Omron Sysmac Studio project Tp last version 30.20h (Comentado) (Sysmac Studio 1.54.0.64019, StandardProject)

# Controller new_Controller_0: NX1P2-9B24DT1 version 1.42
Task PrimaryTask (priority 4, period or condition 4000): Program0
Library OEN_Communication_V1_0_22 1.0.22 (contents left out)

VAR_GLOBAL
    trama : ARRAY[0..4] OF OEN\Modbus\sModbusReq := [(Enable := True, NodeAdr := 1, FunctionCode := Fn15_WriteMultipleCoils, Read := (StartAddressRemote := 0, StartAddressLocal := 0, Count := 0), Write := (StartAddressRemote := 0, StartAddressLocal := 0, Count := 80)), (Enable := True, NodeAdr := 1, FunctionCode := Fn02_ReadDiscreteInputs, Read := (StartAddressRemote := 0, StartAddressLocal := 0, Count := 80), Write := (StartAddressRemote := 0, StartAddressLocal := 0, Count := 0)), (Enable := True, NodeAdr := 1, FunctionCode := Fn04_ReadInputRegisters, Read := (StartAddressRemote := 0, StartAddressLocal := 0, Count := 25), Write := (StartAddressRemote := 0, StartAddressLocal := 0, Count := 0)), (Enable := True, NodeAdr := 1, FunctionCode := Fn16_WriteMultipleRegisters, Read := (StartAddressRemote := 0, StartAddressLocal := 0, Count := 0), Write := (StartAddressRemote := 0, StartAddressLocal := 0, Count := 25)), (Enable := False, NodeAdr := 0, FunctionCode := Fn01_ReadCoils, Read := (StartAddressRemote := 0, StartAddressLocal := 0, Count := 0), Write := (StartAddressRemote := 0, StartAddressLocal := 0, Count := 0))];  (* Trama Responsável pelo invio de informação; published *)
END_VAR
VAR_GLOBAL RETAIN
    Dig_Outputs AT %D10 : ARRAY[0..100] OF BOOL;  (* Digital Outputs; published *)
    Dig_Inputs AT %D20 : ARRAY[0..100] OF BOOL;  (* Digital Inputs; published *)
    Anal_Outputs AT %D30 : ARRAY[0..25] OF WORD;  (* Analog Outputs; published *)
    Anal_Inputs AT %D55 : ARRAY[0..25] OF WORD;  (* Analog Inputs; published *)
END_VAR
VAR_GLOBAL
    Start : BOOL;  (* Acionamento sistema; at BuiltInIO://cpu/#0/Input_Bit_00 *)
    Stop : BOOL;  (* Paragem Sistema; at BuiltInIO://cpu/#0/Input_Bit_01 *)
    ledstart : BOOL;  (* Sinal luminoso de acionamento sistema; at BuiltInIO://cpu/#0/Output_Bit_00 *)
    Colocar : BOOL;  (* Botão Colocar Stacker; at BuiltInIO://cpu/#0/Input_Bit_02 *)
    Remover : BOOL;  (* Botão Remover Stacker; at BuiltInIO://cpu/#0/Input_Bit_03 *)
    NovaCaixa : BOOL;  (* Botão Nova Caixa; at BuiltInIO://cpu/#0/Input_Bit_04 *)
    ledstop : BOOL;  (* Sinal luminoso de paragem sistema; at BuiltInIO://cpu/#0/Output_Bit_01 *)
    ledcolocar : BOOL;  (* Sinal luminoso colocação caixa; at BuiltInIO://cpu/#0/Output_Bit_02 *)
    ledremover : BOOL;  (* Sinal luminoso remoção caixa; at BuiltInIO://cpu/#0/Output_Bit_03 *)
END_VAR

PROGRAM Program0
VAR RETAIN
    Etapas AT %D0 : INT := 0;  (* This variable is change current phase *)
END_VAR
VAR
    Communication_Factory : OEN\Modbus\ModbusTCP_Client;
    Timer2s : TON;
END_VAR
VAR RETAIN
    VariableAux AT %D1 : WORD;  (* Var.aux Medidor Altura 1 *)
END_VAR
VAR
    Timer1 : TON;
    Time_Aux_5 : TIME;  (* Timer_Aux_5s *)
    Timer4 : TON;
    Timer5 : TON;
    Timevariavel : TIME;
    Timer6 : TON;
    Timer10s : TON;
    Timer7 : TON;
    Timer8 : TON;
    Timer9 : TON;
END_VAR
VAR RETAIN
    VariableAux2 : WORD;  (* Var.aux Medidor Altura 1 *)
END_VAR
VAR
    Time_Aux_20 : TIME;  (* Timer_Aux_20s *)
    Timer20 : TON;
    Timer21 : TON;
    Time_Aux_21 : TIME;
    Timer30 : TON;
    Timer31 : TON;
    Timer32 : TON;
    Timer33 : TON;
    Timer34 : TON;
    Timer35 : TON;
    Timer36 : TON;
    Timer37 : TON;
    Timer38 : TON;
    Timer2 : TON;
    Timer2p : TON;
    Timer101 : TON;
    Timer3p : TON;
END_VAR
VAR RETAIN
    VariavelAux10 : WORD;  (* Aux10 *)
END_VAR
VAR
    Timer4sec : TON;
    Timer4P6sec : TON;
    Timer4PPsec : TON;
    Timer5PPsec : TON;
    Timer6PPsec : TON;
    Timer7PPsec : TON;
    Timer8PPsec : TON;
    Timer9PPsec : TON;
    Timer101PPsec : TON;
    Timer10PPsec : TON;
    Timercount : TON;
    Timer3s : TON;
END_VAR
VAR RETAIN
    Count_Caixa_L : INT := 0;  (* Contador Caixa L *)
END_VAR
VAR
    Analogico_L : WORD;  (* Valor Analogico L *)
END_VAR
VAR RETAIN
    Count_Caixa_S : INT := 0;  (* Contador Caixa S *)
END_VAR
VAR
    Analogico_S : WORD;  (* Valor Analogico S *)
END_VAR
VAR RETAIN
    Count_Caixa_M : INT := 0;  (* Contador Caixa M *)
END_VAR
VAR
    Analogico_M : WORD;  (* Valor Analogico M *)
END_VAR
VAR RETAIN
    Contador_Stacker_2 : INT := 0;  (* Contador Posição Stacker 2 *)
    Analogico_Postacker2 : WORD;  (* Variavel Analogica Posição *)
END_VAR
VAR
    Timer30s : TON;
    Timer31s : TON;
    Timer32s : TON;
    TimerEsp : TON;
    TimerDecisão : TON;
    TimerDecisão2 : TON;
    Timerteste : TON;
    led : BOOL;
END_VAR
VAR_EXTERNAL
    trama : ARRAY[0..4] OF OEN\Modbus\sModbusReq;  (* Trama que envia informação *)
    dig_outputs : ARRAY[0..100] OF BOOL;  (* Digital outputs; [8] Tapete 1; [1] Led Botão 1; [2] LED Botão Start; [5] Emissor Caixa; [6] Emissor Paletes 1; [7] Emissor Paletes 2; [11] Tapete 4; [24] Esteira Transportada 11; [14] Tapete Peso (+); [17] Esteira Transportadora 2; [25] Esteira Transportadora 12; [18] Esteira Transportadora 3; [26] Esteira Transportadora 13; [16] Esteira Transportadora 1; [10] Tapete 3; [33] Two-Axis Pick &amp; Place 1 Z; [36] Two-Axis Pick &amp; Place 1 (Grab); [38] Two-Axis Pick &amp; Place 1 Rotate CW; [9] Tapete 2; [32] Two-Axis Pick &amp; Place 1 X; [41] Two-Axis Pick &amp; Place 1 Rotate CCW; [19] Esteira Transportadora 4; [20] Esteira Transportadora 5; [21] Esteira Transportadora 6; [22] Esteira Transportadora 7; [23] Esteira Transportadora 8; [30] pusher 1; [12] Tapete 5; [15] Tapete peso 2; [13] Tapete 6; [49] Stacker Crane 3(left); [47] Stacker Crane 3 lift; [54] Led Colocar; [51] Stacker Crane 3 Right ; [55] LED Remover; [53] Remover 3; [35] Two-Axis Pick &amp; Place 2 Z; [37] Two-Axis Pick &amp; Place 2 (Grab); [39] Two-Axis Pick &amp; Place 2 Rotate CW; [34] Two-Axis Pick &amp; Place 2 X; [43] Two-Axis Pick &amp; Place 1 Rotate CCW; [27] Esteira Transportadora 14; [28] Esteira Transportadora 15; [29] Esteira Transportadora 16; [31] Pusher 2; [48] Stacker Crane 1 left; [46] Stacker Crane 1 lift; [50] stacker crane 1 right; [3] LED Botão Stop *)
    dig_inputs : ARRAY[0..100] OF BOOL;  (* Digital inputs; [2] Sensor Detetar caixas; [0] Botão Start; [13] Sensor Difuso 10; [22] Sensor Difuso 19; [3] Sensor Difuso 1; [14] Sensor Difuso 11; [9] Sensor Difuso 6; [21] Sensor difuso 18; [15] Sensor Difuso 12; [16] Sensor difuso 13; [59] Sensor Difuso 27; [23] Sensor Difuso 20; [24] Sensor Difuso 21; [4] Sensor Difuso 2; [5] Sensor Difuso 3; [52] Two-Axis Pick &amp; Place 1 (Moving Z); [36] Two-Axis Pick &amp; Place 1 (Grab); [50] Two-Axis Pick &amp; Place 1 (Detected); [17] Sensor difuso 14; [18] Sensor difuso 15; [19] sensor difuso 16; [20] Sensor Difuso 17; [35] Pusher frontal; [7] Sensor Difuso 4; [8] Sensor Difuso 8; [60] Sensor Difuso 28; [29] Sensor Refletivo 1; [61] Botão Colocar; [44] Stacker Crane 3 left limit; [48] Stacker Crane 3 Middle Limit; [46] Stacker Crane 3 Right Limit; [62] Botão Remover; [31] Sensor Refletivo 3; [30] Sensor Difuso 29; [10] Sensor difuso 7; [12] Sensor Difuso 9; [26] Sensor Difuso 23; [27] Sensor Difuso 24; [32] Sensor Refletivo 4; [28] Sensor Difuso 25; [11] Sensor Difuso 8; [54] detected; [43] Stacker Crane 1 left Limit; [47] stacker Crane 1 Middle Limit; [45] Stacker Crane 1 Right Limit; [1] Botão Stop; [63] Botão Nova Caixa *)
    anal_inputs : ARRAY[0..25] OF WORD;  (* Analog inputs; [2] Balança 1 Peso (V); [1] Medidor Altura 2; [0] Medidor Altura 1; [3] Peso 2 *)
    anal_outputs : ARRAY[0..25] OF WORD;  (* Analog outputs; [2] Esteira Transportadora 9; [10] Display 1; [12] Display 3; [1] Posição 2; [11] Display 2; [6] Loading Convoyer 1; [0] Posição1 *)
    Start : BOOL;
    Stop : BOOL;
    ledstart : BOOL;
    ledstop : BOOL;
    NovaCaixa : BOOL;
    Colocar : BOOL;
    Remover : BOOL;
    ledremover : BOOL;
    ledcolocar : BOOL;
END_VAR
VAR
    _p1 : BOOL;
    _e2 : R_TRIG;
    _p3 : BOOL;
    _p4 : BOOL;
    _p5 : BOOL;
    _e6 : R_TRIG;
    _e7 : R_TRIG;
    _e8 : R_TRIG;
END_VAR

(* Section Phases: ladder, written here as Structured Text *)

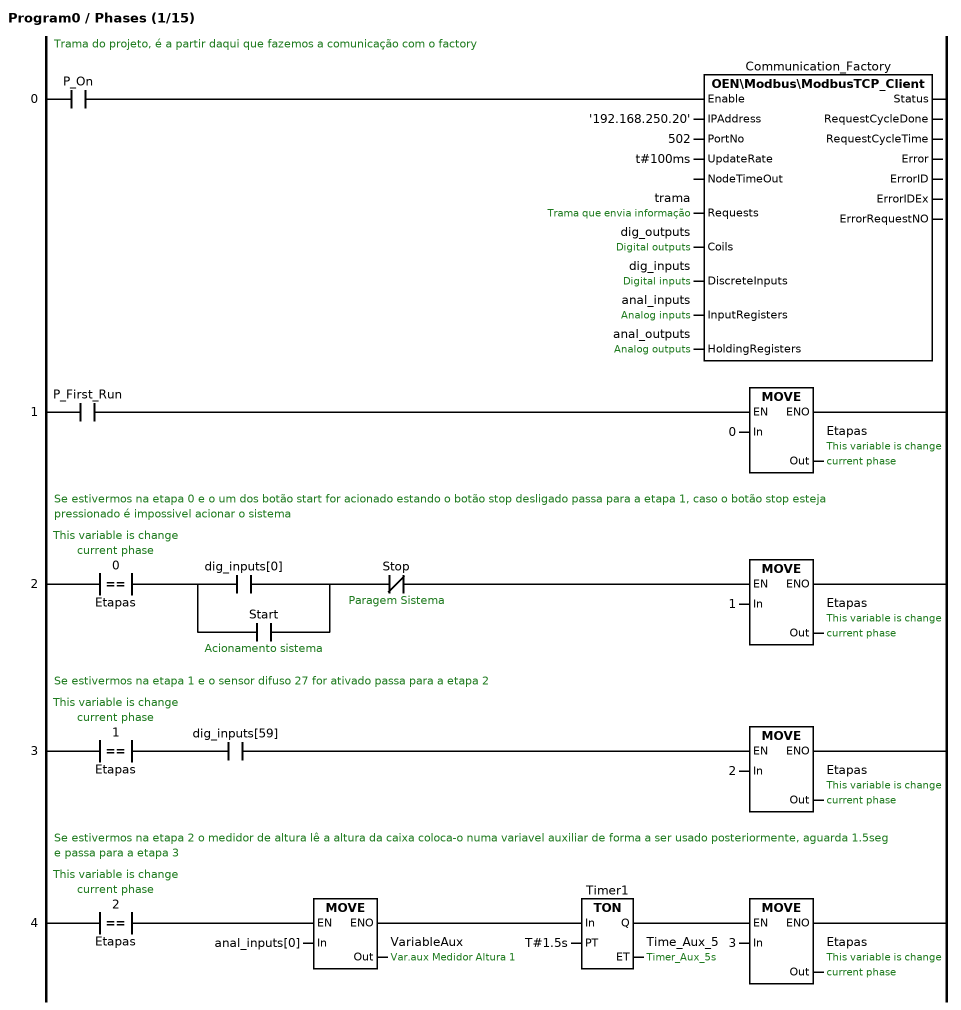
(* Rung 0: Trama do projeto, é a partir daqui que fazemos a comunicação com o factory *)
Communication_Factory(Enable := P_On, IPAddress := '192.168.250.20', PortNo := 502, UpdateRate := t#100ms, Requests := trama, Coils := dig_outputs, DiscreteInputs := dig_inputs, InputRegisters := anal_inputs, HoldingRegisters := anal_outputs);
(* Rung 1 *)
IF P_First_Run THEN Etapas := 0; END_IF;
(* Rung 2: Se estivermos na etapa 0 e o um dos botão start for acionado estando o botão stop desligado passa para a etapa 1, caso o botão stop esteja pressionado é impossivel acionar o sistema *)
IF (0 = Etapas) AND (dig_inputs[0] OR Start) AND NOT Stop THEN Etapas := 1; END_IF;
(* Rung 3: Se estivermos na etapa 1 e o sensor difuso 27 for ativado passa para a etapa 2 *)
IF (1 = Etapas) AND dig_inputs[59] THEN Etapas := 2; END_IF;
(* Rung 4: Se estivermos na etapa 2 o medidor de altura lê a altura da caixa coloca-o numa variavel auxiliar de forma a ser usado posteriormente, aguarda 1.5seg e passa para a etapa 3 *)
IF 2 = Etapas THEN VariableAux := anal_inputs[0]; END_IF;
Timer1(In := 2 = Etapas, PT := T#1.5s, ET => Time_Aux_5);
IF Timer1.Q THEN Etapas := 3; END_IF;

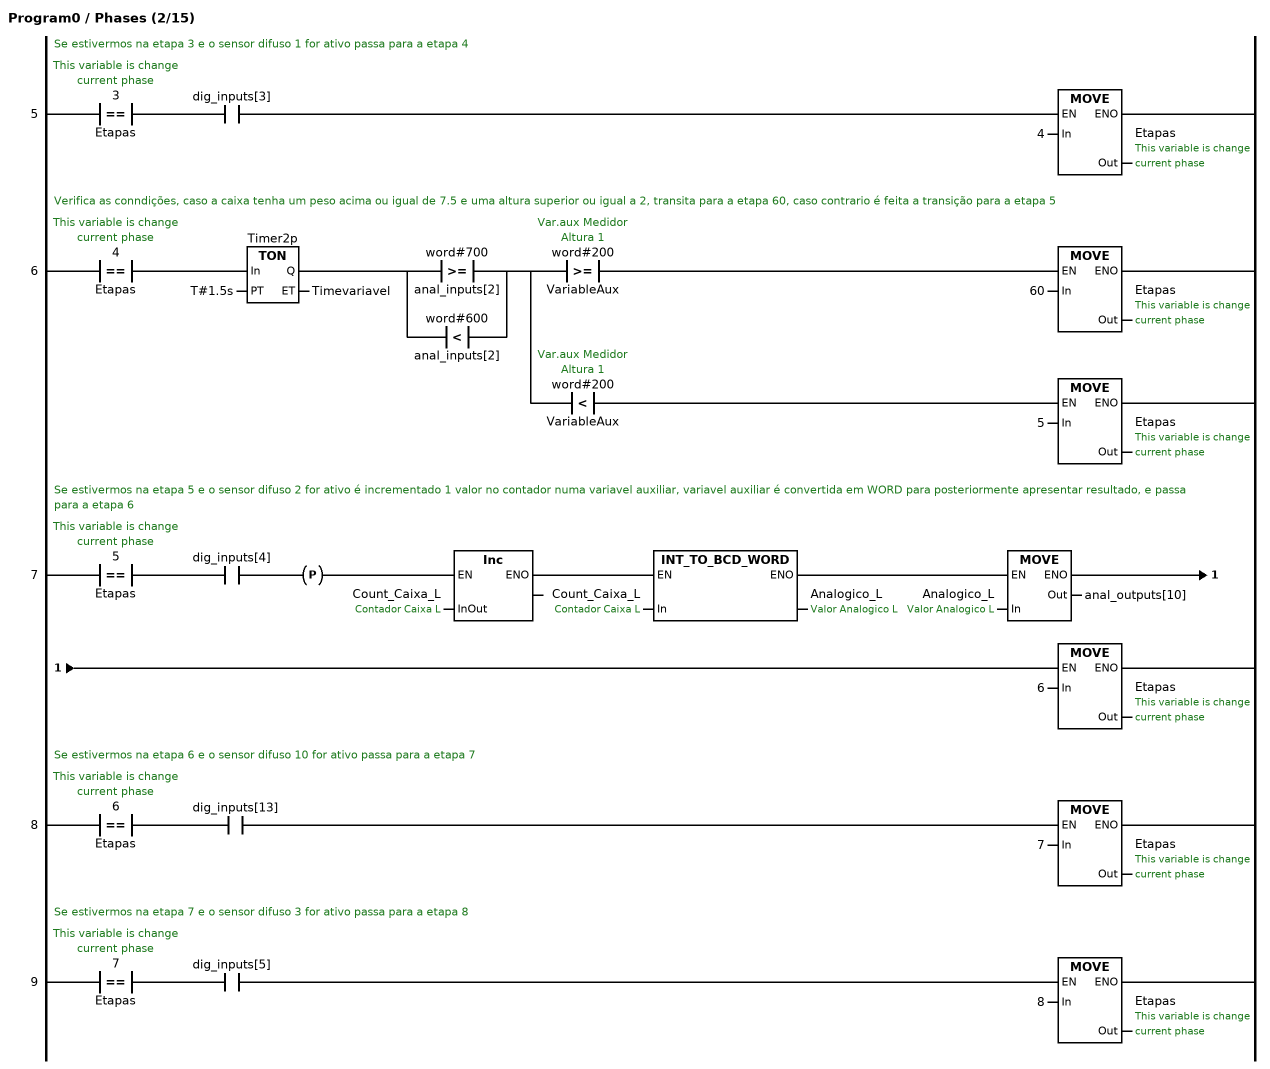
(* Rung 5: Se estivermos na etapa 3 e o sensor difuso 1 for ativo passa para a etapa 4 *)
IF (3 = Etapas) AND dig_inputs[3] THEN Etapas := 4; END_IF;
(* Rung 6: Verifica as conndições, caso a caixa tenha um peso acima ou igual de 7.5 e uma altura superior ou igual a 2, transita para a etapa 60, caso contrario é feita a transição para a etapa 5 *)
Timer2p(In := 4 = Etapas, PT := T#1.5s, ET => Timevariavel);
_p1 := Timer2p.Q AND ((word#700 >= anal_inputs[2]) OR (word#600 < anal_inputs[2]));
IF _p1 AND (word#200 >= VariableAux) THEN Etapas := 60; END_IF;
IF _p1 AND (word#200 < VariableAux) THEN Etapas := 5; END_IF;
(* Rung 7: Se estivermos na etapa 5 e o sensor difuso 2 for ativo é incrementado 1 valor no contador numa variavel auxiliar, variavel auxiliar é convertida em WORD para posteriormente apresentar resultado, e passa para a etapa 6 *)
_e2(CLK := (5 = Etapas) AND dig_inputs[4]);
IF _e2.Q THEN
    Inc(InOut := Count_Caixa_L);
    Analogico_L := INT_TO_BCD_WORD(In := Count_Caixa_L);
    anal_outputs[10] := Analogico_L;
    Etapas := 6;
END_IF;
(* Rung 8: Se estivermos na etapa 6 e o sensor difuso 10 for ativo passa para a etapa 7 *)
IF (6 = Etapas) AND dig_inputs[13] THEN Etapas := 7; END_IF;
(* Rung 9: Se estivermos na etapa 7 e o sensor difuso 3 for ativo passa para a etapa 8 *)
IF (7 = Etapas) AND dig_inputs[5] THEN Etapas := 8; END_IF;

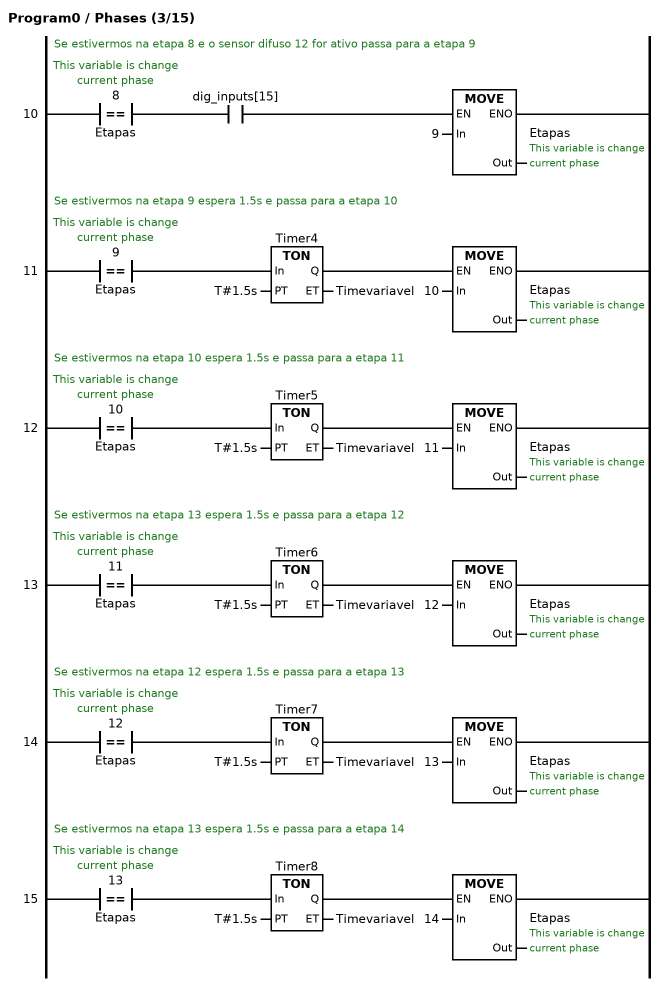
(* Rung 10: Se estivermos na etapa 8 e o sensor difuso 12 for ativo passa para a etapa 9 *)
IF (8 = Etapas) AND dig_inputs[15] THEN Etapas := 9; END_IF;
(* Rung 11: Se estivermos na etapa 9 espera 1.5s e passa para a etapa 10 *)
Timer4(In := 9 = Etapas, PT := T#1.5s, ET => Timevariavel);
IF Timer4.Q THEN Etapas := 10; END_IF;
(* Rung 12: Se estivermos na etapa 10 espera 1.5s e passa para a etapa 11 *)
Timer5(In := 10 = Etapas, PT := T#1.5s, ET => Timevariavel);
IF Timer5.Q THEN Etapas := 11; END_IF;
(* Rung 13: Se estivermos na etapa 13 espera 1.5s e passa para a etapa 12 *)
Timer6(In := 11 = Etapas, PT := T#1.5s, ET => Timevariavel);
IF Timer6.Q THEN Etapas := 12; END_IF;
(* Rung 14: Se estivermos na etapa 12 espera 1.5s e passa para a etapa 13 *)
Timer7(In := 12 = Etapas, PT := T#1.5s, ET => Timevariavel);
IF Timer7.Q THEN Etapas := 13; END_IF;
(* Rung 15: Se estivermos na etapa 13 espera 1.5s e passa para a etapa 14 *)
Timer8(In := 13 = Etapas, PT := T#1.5s, ET => Timevariavel);
IF Timer8.Q THEN Etapas := 14; END_IF;

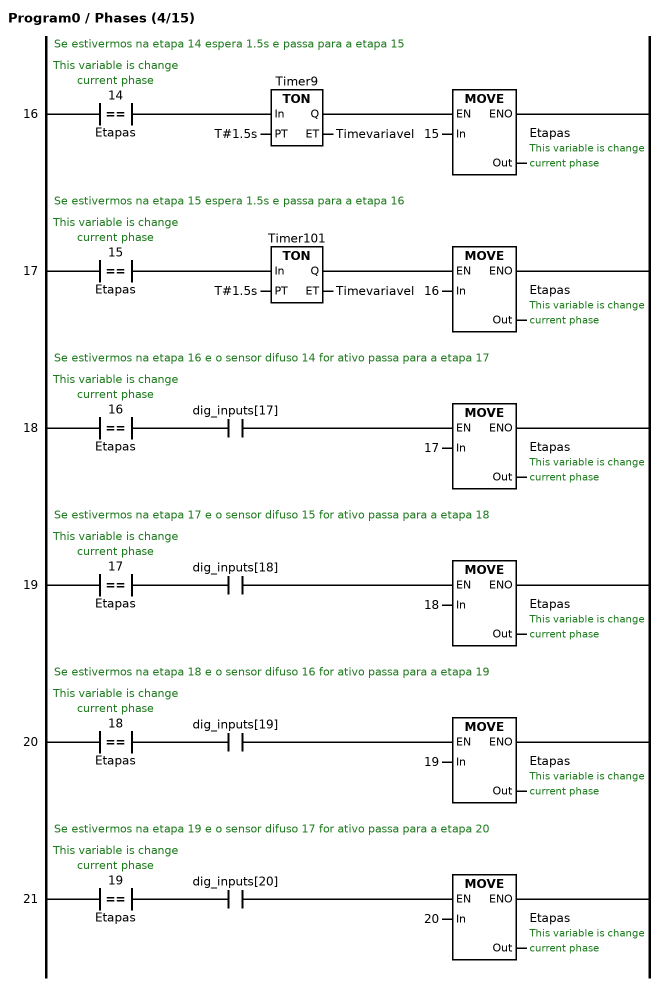
(* Rung 16: Se estivermos na etapa 14 espera 1.5s e passa para a etapa 15 *)
Timer9(In := 14 = Etapas, PT := T#1.5s, ET => Timevariavel);
IF Timer9.Q THEN Etapas := 15; END_IF;
(* Rung 17: Se estivermos na etapa 15 espera 1.5s e passa para a etapa 16 *)
Timer101(In := 15 = Etapas, PT := T#1.5s, ET => Timevariavel);
IF Timer101.Q THEN Etapas := 16; END_IF;
(* Rung 18: Se estivermos na etapa 16 e o sensor difuso 14 for ativo passa para a etapa 17 *)
IF (16 = Etapas) AND dig_inputs[17] THEN Etapas := 17; END_IF;
(* Rung 19: Se estivermos na etapa 17 e o sensor difuso 15 for ativo passa para a etapa 18 *)
IF (17 = Etapas) AND dig_inputs[18] THEN Etapas := 18; END_IF;
(* Rung 20: Se estivermos na etapa 18 e o sensor difuso 16 for ativo passa para a etapa 19 *)
IF (18 = Etapas) AND dig_inputs[19] THEN Etapas := 19; END_IF;
(* Rung 21: Se estivermos na etapa 19 e o sensor difuso 17 for ativo passa para a etapa 20 *)
IF (19 = Etapas) AND dig_inputs[20] THEN Etapas := 20; END_IF;

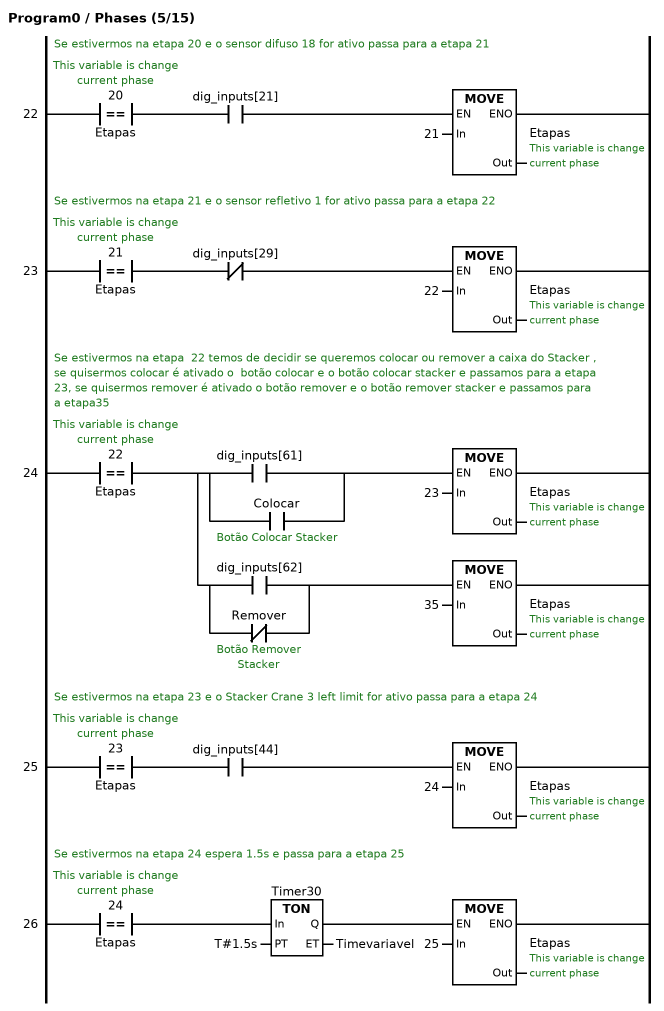
(* Rung 22: Se estivermos na etapa 20 e o sensor difuso 18 for ativo passa para a etapa 21 *)
IF (20 = Etapas) AND dig_inputs[21] THEN Etapas := 21; END_IF;
(* Rung 23: Se estivermos na etapa 21 e o sensor refletivo 1 for ativo passa para a etapa 22 *)
IF (21 = Etapas) AND NOT dig_inputs[29] THEN Etapas := 22; END_IF;
(* Rung 24: Se estivermos na etapa  22 temos de decidir se queremos colocar ou remover a caixa do Stacker , se quisermos colocar é ativado o  botão colocar e o botão colocar stacker e passamos para a etapa 23, se quisermos remover é ativado o botão remover e o botão remover stacker e passamos para a etapa35 *)
_p3 := 22 = Etapas;
IF (22 = Etapas) AND (dig_inputs[61] OR Colocar) THEN Etapas := 23; END_IF;
IF _p3 AND (dig_inputs[62] OR NOT Remover) THEN Etapas := 35; END_IF;
(* Rung 25: Se estivermos na etapa 23 e o Stacker Crane 3 left limit for ativo passa para a etapa 24 *)
IF (23 = Etapas) AND dig_inputs[44] THEN Etapas := 24; END_IF;
(* Rung 26: Se estivermos na etapa 24 espera 1.5s e passa para a etapa 25 *)
Timer30(In := 24 = Etapas, PT := T#1.5s, ET => Timevariavel);
IF Timer30.Q THEN Etapas := 25; END_IF;

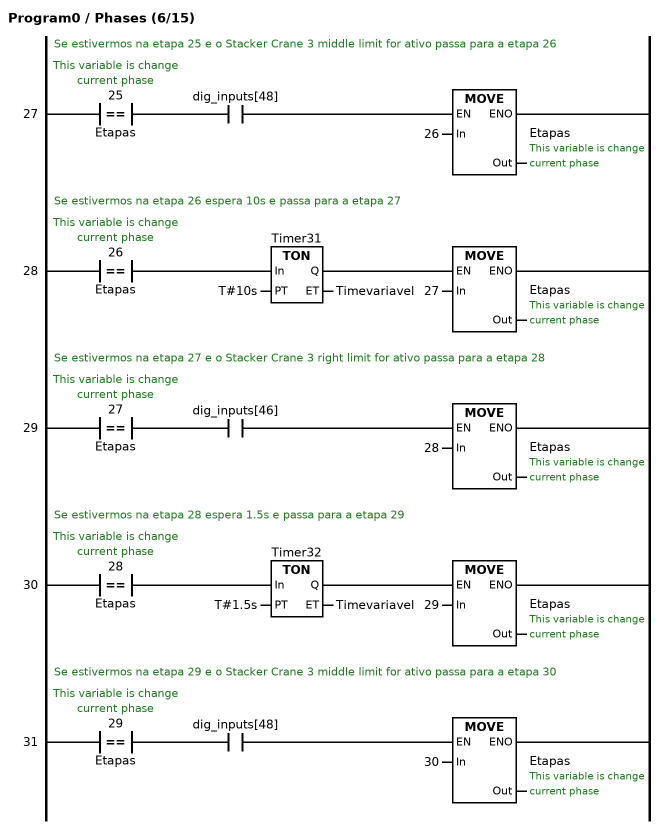
(* Rung 27: Se estivermos na etapa 25 e o Stacker Crane 3 middle limit for ativo passa para a etapa 26 *)
IF (25 = Etapas) AND dig_inputs[48] THEN Etapas := 26; END_IF;
(* Rung 28: Se estivermos na etapa 26 espera 10s e passa para a etapa 27 *)
Timer31(In := 26 = Etapas, PT := T#10s, ET => Timevariavel);
IF Timer31.Q THEN Etapas := 27; END_IF;
(* Rung 29: Se estivermos na etapa 27 e o Stacker Crane 3 right limit for ativo passa para a etapa 28 *)
IF (27 = Etapas) AND dig_inputs[46] THEN Etapas := 28; END_IF;
(* Rung 30: Se estivermos na etapa 28 espera 1.5s e passa para a etapa 29 *)
Timer32(In := 28 = Etapas, PT := T#1.5s, ET => Timevariavel);
IF Timer32.Q THEN Etapas := 29; END_IF;
(* Rung 31: Se estivermos na etapa 29 e o Stacker Crane 3 middle limit for ativo passa para a etapa 30 *)
IF (29 = Etapas) AND dig_inputs[48] THEN Etapas := 30; END_IF;

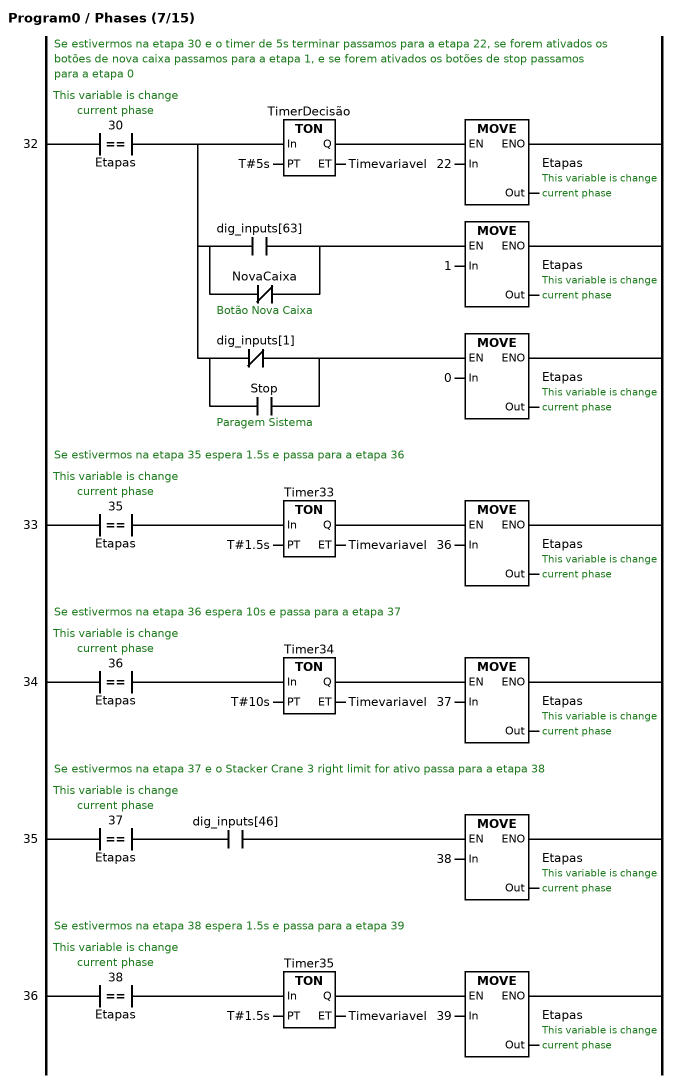
(* Rung 32: Se estivermos na etapa 30 e o timer de 5s terminar passamos para a etapa 22, se forem ativados os botões de nova caixa passamos para a etapa 1, e se forem ativados os botões de stop passamos para a etapa 0 *)
TimerDecisão(In := 30 = Etapas, PT := T#5s, ET => Timevariavel);
_p4 := 30 = Etapas;
IF TimerDecisão.Q THEN Etapas := 22; END_IF;
IF _p4 AND (dig_inputs[63] OR NOT NovaCaixa) THEN Etapas := 1; END_IF;
IF _p4 AND (NOT dig_inputs[1] OR Stop) THEN Etapas := 0; END_IF;
(* Rung 33: Se estivermos na etapa 35 espera 1.5s e passa para a etapa 36 *)
Timer33(In := 35 = Etapas, PT := T#1.5s, ET => Timevariavel);
IF Timer33.Q THEN Etapas := 36; END_IF;
(* Rung 34: Se estivermos na etapa 36 espera 10s e passa para a etapa 37 *)
Timer34(In := 36 = Etapas, PT := T#10s, ET => Timevariavel);
IF Timer34.Q THEN Etapas := 37; END_IF;
(* Rung 35: Se estivermos na etapa 37 e o Stacker Crane 3 right limit for ativo passa para a etapa 38 *)
IF (37 = Etapas) AND dig_inputs[46] THEN Etapas := 38; END_IF;
(* Rung 36: Se estivermos na etapa 38 espera 1.5s e passa para a etapa 39 *)
Timer35(In := 38 = Etapas, PT := T#1.5s, ET => Timevariavel);
IF Timer35.Q THEN Etapas := 39; END_IF;

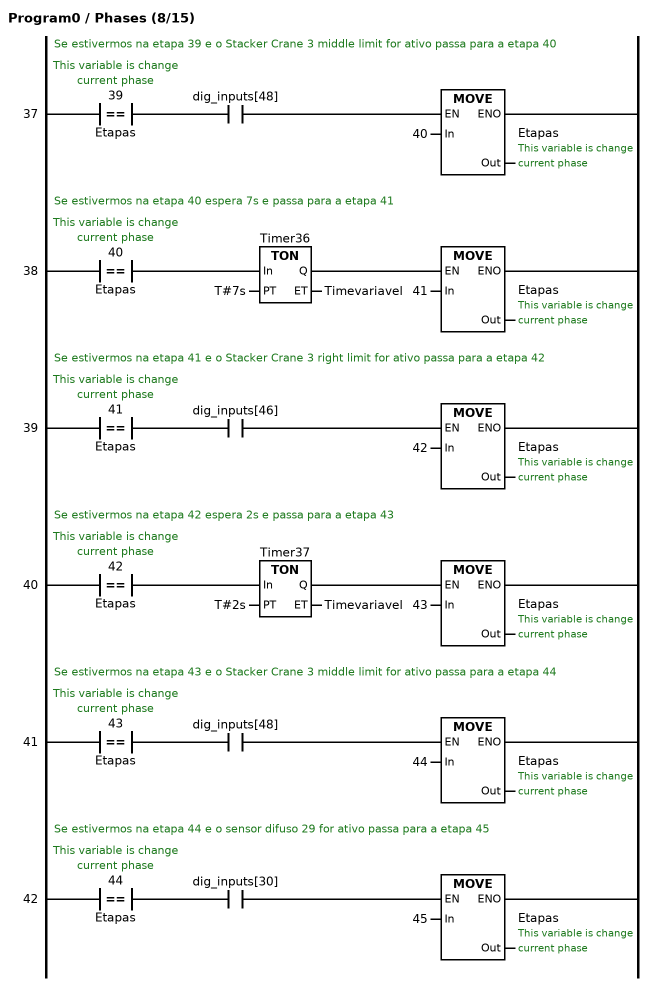
(* Rung 37: Se estivermos na etapa 39 e o Stacker Crane 3 middle limit for ativo passa para a etapa 40 *)
IF (39 = Etapas) AND dig_inputs[48] THEN Etapas := 40; END_IF;
(* Rung 38: Se estivermos na etapa 40 espera 7s e passa para a etapa 41 *)
Timer36(In := 40 = Etapas, PT := T#7s, ET => Timevariavel);
IF Timer36.Q THEN Etapas := 41; END_IF;
(* Rung 39: Se estivermos na etapa 41 e o Stacker Crane 3 right limit for ativo passa para a etapa 42 *)
IF (41 = Etapas) AND dig_inputs[46] THEN Etapas := 42; END_IF;
(* Rung 40: Se estivermos na etapa 42 espera 2s e passa para a etapa 43 *)
Timer37(In := 42 = Etapas, PT := T#2s, ET => Timevariavel);
IF Timer37.Q THEN Etapas := 43; END_IF;
(* Rung 41: Se estivermos na etapa 43 e o Stacker Crane 3 middle limit for ativo passa para a etapa 44 *)
IF (43 = Etapas) AND dig_inputs[48] THEN Etapas := 44; END_IF;
(* Rung 42: Se estivermos na etapa 44 e o sensor difuso 29 for ativo passa para a etapa 45 *)
IF (44 = Etapas) AND dig_inputs[30] THEN Etapas := 45; END_IF;

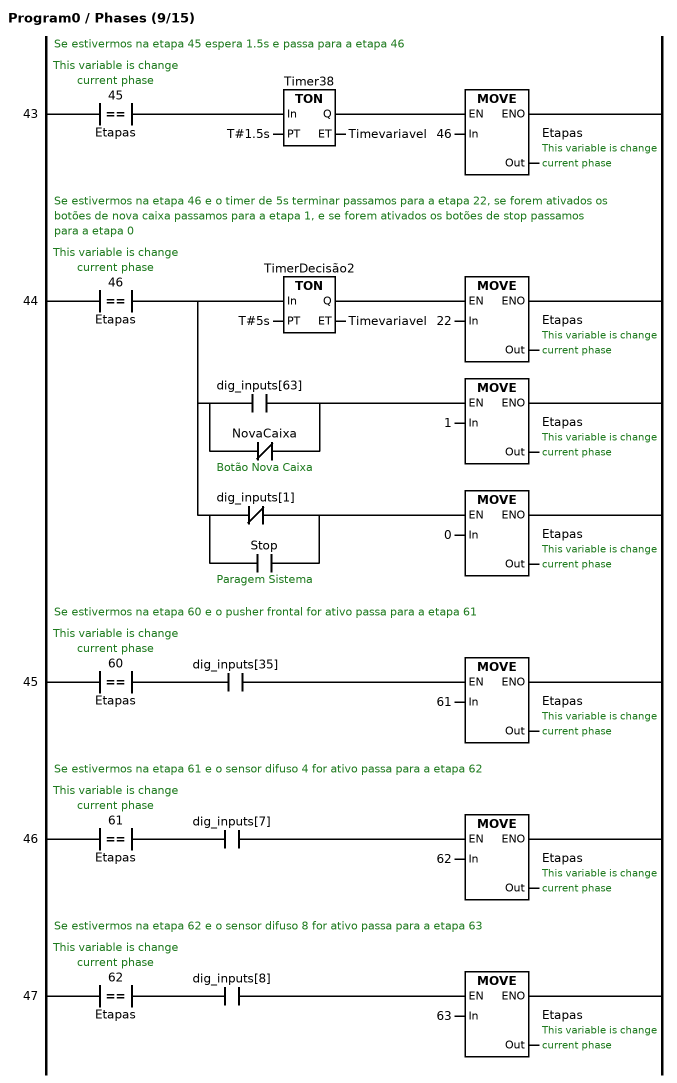
(* Rung 43: Se estivermos na etapa 45 espera 1.5s e passa para a etapa 46 *)
Timer38(In := 45 = Etapas, PT := T#1.5s, ET => Timevariavel);
IF Timer38.Q THEN Etapas := 46; END_IF;
(* Rung 44: Se estivermos na etapa 46 e o timer de 5s terminar passamos para a etapa 22, se forem ativados os botões de nova caixa passamos para a etapa 1, e se forem ativados os botões de stop passamos para a etapa 0 *)
TimerDecisão2(In := 46 = Etapas, PT := T#5s, ET => Timevariavel);
_p5 := 46 = Etapas;
IF TimerDecisão2.Q THEN Etapas := 22; END_IF;
IF _p5 AND (dig_inputs[63] OR NOT NovaCaixa) THEN Etapas := 1; END_IF;
IF _p5 AND (NOT dig_inputs[1] OR Stop) THEN Etapas := 0; END_IF;
(* Rung 45: Se estivermos na etapa 60 e o pusher frontal for ativo passa para a etapa 61 *)
IF (60 = Etapas) AND dig_inputs[35] THEN Etapas := 61; END_IF;
(* Rung 46: Se estivermos na etapa 61 e o sensor difuso 4 for ativo passa para a etapa 62 *)
IF (61 = Etapas) AND dig_inputs[7] THEN Etapas := 62; END_IF;
(* Rung 47: Se estivermos na etapa 62 e o sensor difuso 8 for ativo passa para a etapa 63 *)
IF (62 = Etapas) AND dig_inputs[8] THEN Etapas := 63; END_IF;

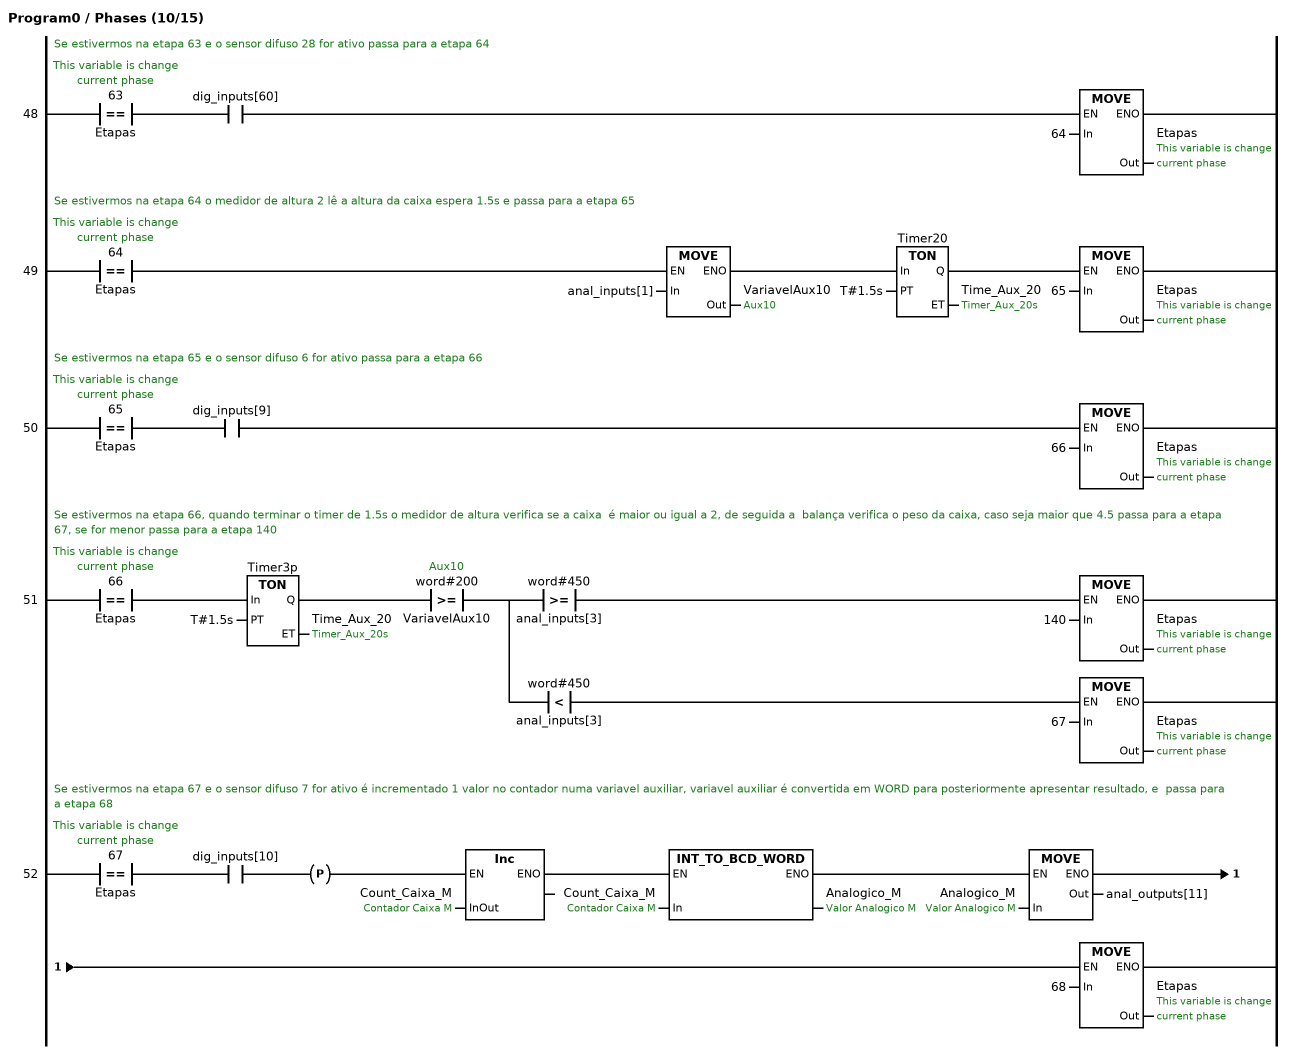
(* Rung 48: Se estivermos na etapa 63 e o sensor difuso 28 for ativo passa para a etapa 64 *)
IF (63 = Etapas) AND dig_inputs[60] THEN Etapas := 64; END_IF;
(* Rung 49: Se estivermos na etapa 64 o medidor de altura 2 lê a altura da caixa espera 1.5s e passa para a etapa 65 *)
IF 64 = Etapas THEN VariavelAux10 := anal_inputs[1]; END_IF;
Timer20(In := 64 = Etapas, PT := T#1.5s, ET => Time_Aux_20);
IF Timer20.Q THEN Etapas := 65; END_IF;
(* Rung 50: Se estivermos na etapa 65 e o sensor difuso 6 for ativo passa para a etapa 66 *)
IF (65 = Etapas) AND dig_inputs[9] THEN Etapas := 66; END_IF;
(* Rung 51: Se estivermos na etapa 66, quando terminar o timer de 1.5s o medidor de altura verifica se a caixa  é maior ou igual a 2, de seguida a  balança verifica o peso da caixa, caso seja maior que 4.5 passa para a etapa 67, se for menor passa para a etapa 140 *)
Timer3p(In := 66 = Etapas, PT := T#1.5s, ET => Time_Aux_20);
IF Timer3p.Q AND (word#200 >= VariavelAux10) AND (word#450 >= anal_inputs[3]) THEN Etapas := 140; END_IF;
IF Timer3p.Q AND (word#200 >= VariavelAux10) AND (word#450 < anal_inputs[3]) THEN Etapas := 67; END_IF;
(* Rung 52: Se estivermos na etapa 67 e o sensor difuso 7 for ativo é incrementado 1 valor no contador numa variavel auxiliar, variavel auxiliar é convertida em WORD para posteriormente apresentar resultado, e  passa para a etapa 68 *)
_e6(CLK := (67 = Etapas) AND dig_inputs[10]);
IF _e6.Q THEN
    Inc(InOut := Count_Caixa_M);
    Analogico_M := INT_TO_BCD_WORD(In := Count_Caixa_M);
    anal_outputs[11] := Analogico_M;
    Etapas := 68;
END_IF;

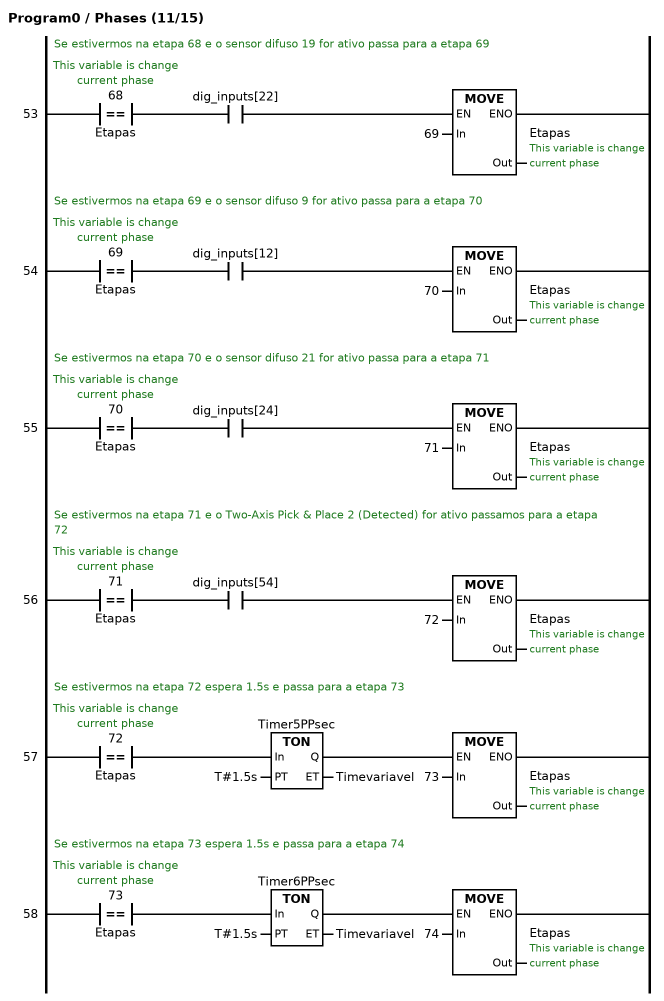
(* Rung 53: Se estivermos na etapa 68 e o sensor difuso 19 for ativo passa para a etapa 69 *)
IF (68 = Etapas) AND dig_inputs[22] THEN Etapas := 69; END_IF;
(* Rung 54: Se estivermos na etapa 69 e o sensor difuso 9 for ativo passa para a etapa 70 *)
IF (69 = Etapas) AND dig_inputs[12] THEN Etapas := 70; END_IF;
(* Rung 55: Se estivermos na etapa 70 e o sensor difuso 21 for ativo passa para a etapa 71 *)
IF (70 = Etapas) AND dig_inputs[24] THEN Etapas := 71; END_IF;
(* Rung 56: Se estivermos na etapa 71 e o Two-Axis Pick & Place 2 (Detected) for ativo passamos para a etapa 72 *)
IF (71 = Etapas) AND dig_inputs[54] THEN Etapas := 72; END_IF;
(* Rung 57: Se estivermos na etapa 72 espera 1.5s e passa para a etapa 73 *)
Timer5PPsec(In := 72 = Etapas, PT := T#1.5s, ET => Timevariavel);
IF Timer5PPsec.Q THEN Etapas := 73; END_IF;
(* Rung 58: Se estivermos na etapa 73 espera 1.5s e passa para a etapa 74 *)
Timer6PPsec(In := 73 = Etapas, PT := T#1.5s, ET => Timevariavel);
IF Timer6PPsec.Q THEN Etapas := 74; END_IF;

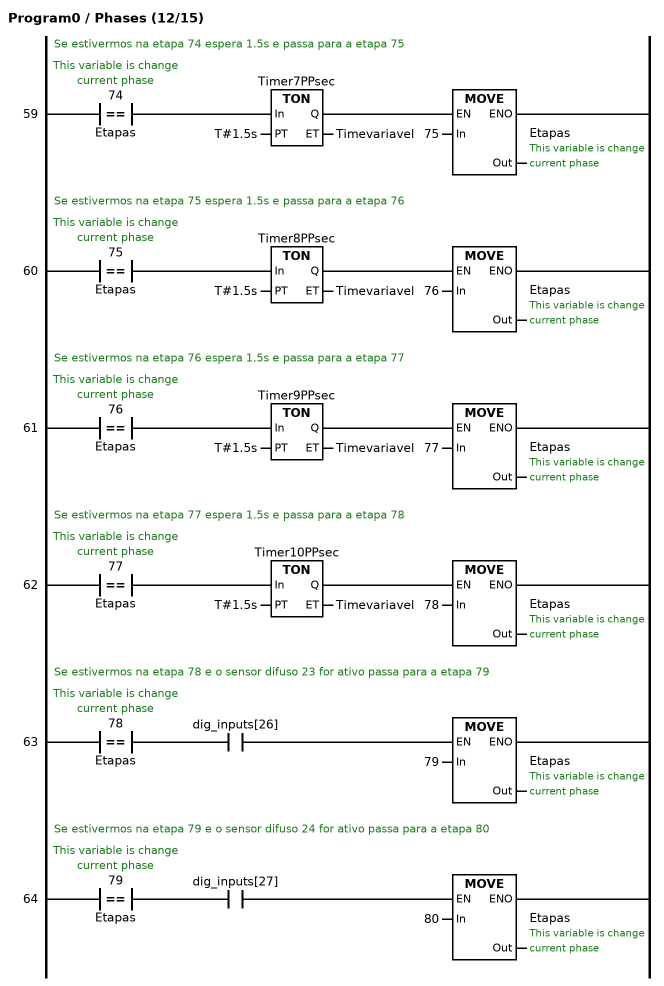
(* Rung 59: Se estivermos na etapa 74 espera 1.5s e passa para a etapa 75 *)
Timer7PPsec(In := 74 = Etapas, PT := T#1.5s, ET => Timevariavel);
IF Timer7PPsec.Q THEN Etapas := 75; END_IF;
(* Rung 60: Se estivermos na etapa 75 espera 1.5s e passa para a etapa 76 *)
Timer8PPsec(In := 75 = Etapas, PT := T#1.5s, ET => Timevariavel);
IF Timer8PPsec.Q THEN Etapas := 76; END_IF;
(* Rung 61: Se estivermos na etapa 76 espera 1.5s e passa para a etapa 77 *)
Timer9PPsec(In := 76 = Etapas, PT := T#1.5s, ET => Timevariavel);
IF Timer9PPsec.Q THEN Etapas := 77; END_IF;
(* Rung 62: Se estivermos na etapa 77 espera 1.5s e passa para a etapa 78 *)
Timer10PPsec(In := 77 = Etapas, PT := T#1.5s, ET => Timevariavel);
IF Timer10PPsec.Q THEN Etapas := 78; END_IF;
(* Rung 63: Se estivermos na etapa 78 e o sensor difuso 23 for ativo passa para a etapa 79 *)
IF (78 = Etapas) AND dig_inputs[26] THEN Etapas := 79; END_IF;
(* Rung 64: Se estivermos na etapa 79 e o sensor difuso 24 for ativo passa para a etapa 80 *)
IF (79 = Etapas) AND dig_inputs[27] THEN Etapas := 80; END_IF;

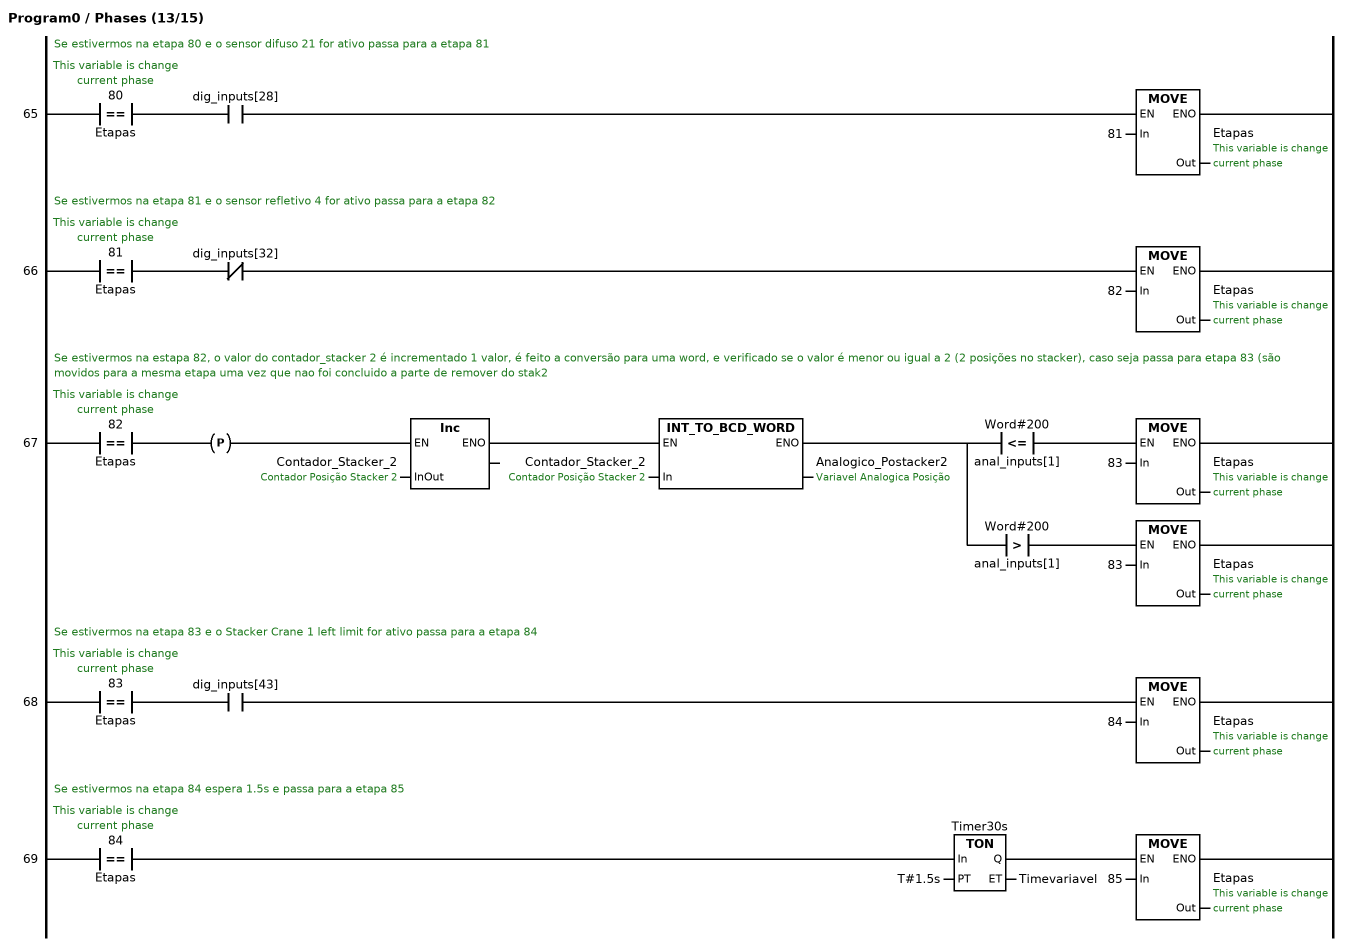
(* Rung 65: Se estivermos na etapa 80 e o sensor difuso 21 for ativo passa para a etapa 81 *)
IF (80 = Etapas) AND dig_inputs[28] THEN Etapas := 81; END_IF;
(* Rung 66: Se estivermos na etapa 81 e o sensor refletivo 4 for ativo passa para a etapa 82 *)
IF (81 = Etapas) AND NOT dig_inputs[32] THEN Etapas := 82; END_IF;
(* Rung 67: Se estivermos na estapa 82, o valor do contador_stacker 2 é incrementado 1 valor, é feito a conversão para uma word, e verificado se o valor é menor ou igual a 2 (2 posições no stacker), caso seja passa para etapa 83 (são movidos para a mesma etapa uma vez que nao foi concluido a parte de remover do stak2 *)
_e7(CLK := 82 = Etapas);
IF _e7.Q THEN
    Inc(InOut := Contador_Stacker_2);
    Analogico_Postacker2 := INT_TO_BCD_WORD(In := Contador_Stacker_2);
END_IF;
IF _e7.Q AND (Word#200 <= anal_inputs[1]) THEN Etapas := 83; END_IF;
IF _e7.Q AND (Word#200 > anal_inputs[1]) THEN Etapas := 83; END_IF;
(* Rung 68: Se estivermos na etapa 83 e o Stacker Crane 1 left limit for ativo passa para a etapa 84 *)
IF (83 = Etapas) AND dig_inputs[43] THEN Etapas := 84; END_IF;
(* Rung 69: Se estivermos na etapa 84 espera 1.5s e passa para a etapa 85 *)
Timer30s(In := 84 = Etapas, PT := T#1.5s, ET => Timevariavel);
IF Timer30s.Q THEN Etapas := 85; END_IF;

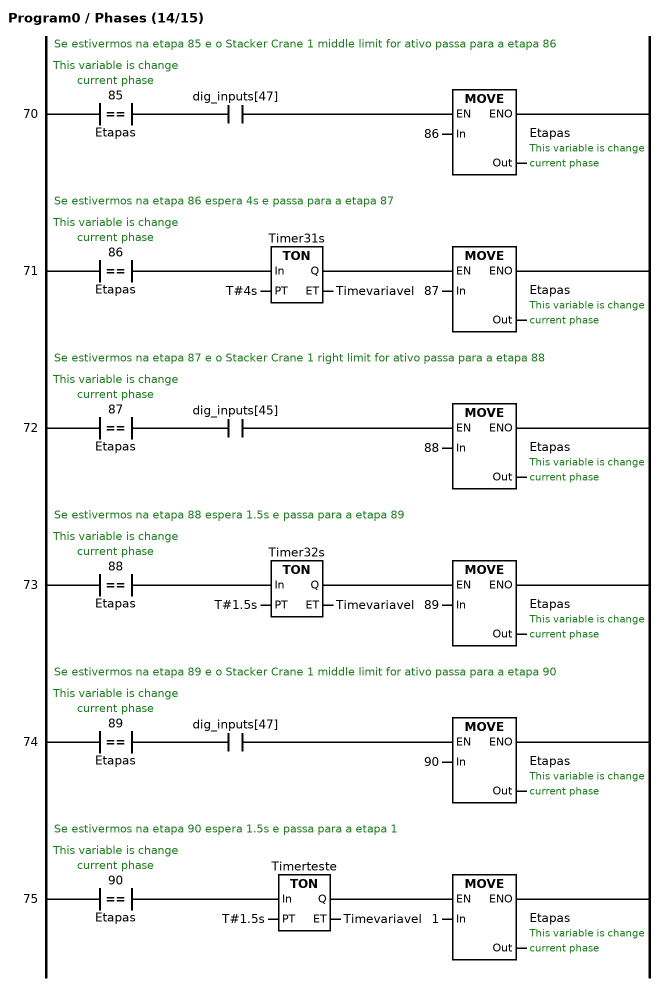
(* Rung 70: Se estivermos na etapa 85 e o Stacker Crane 1 middle limit for ativo passa para a etapa 86 *)
IF (85 = Etapas) AND dig_inputs[47] THEN Etapas := 86; END_IF;
(* Rung 71: Se estivermos na etapa 86 espera 4s e passa para a etapa 87 *)
Timer31s(In := 86 = Etapas, PT := T#4s, ET => Timevariavel);
IF Timer31s.Q THEN Etapas := 87; END_IF;
(* Rung 72: Se estivermos na etapa 87 e o Stacker Crane 1 right limit for ativo passa para a etapa 88 *)
IF (87 = Etapas) AND dig_inputs[45] THEN Etapas := 88; END_IF;
(* Rung 73: Se estivermos na etapa 88 espera 1.5s e passa para a etapa 89 *)
Timer32s(In := 88 = Etapas, PT := T#1.5s, ET => Timevariavel);
IF Timer32s.Q THEN Etapas := 89; END_IF;
(* Rung 74: Se estivermos na etapa 89 e o Stacker Crane 1 middle limit for ativo passa para a etapa 90 *)
IF (89 = Etapas) AND dig_inputs[47] THEN Etapas := 90; END_IF;
(* Rung 75: Se estivermos na etapa 90 espera 1.5s e passa para a etapa 1 *)
Timerteste(In := 90 = Etapas, PT := T#1.5s, ET => Timevariavel);
IF Timerteste.Q THEN Etapas := 1; END_IF;

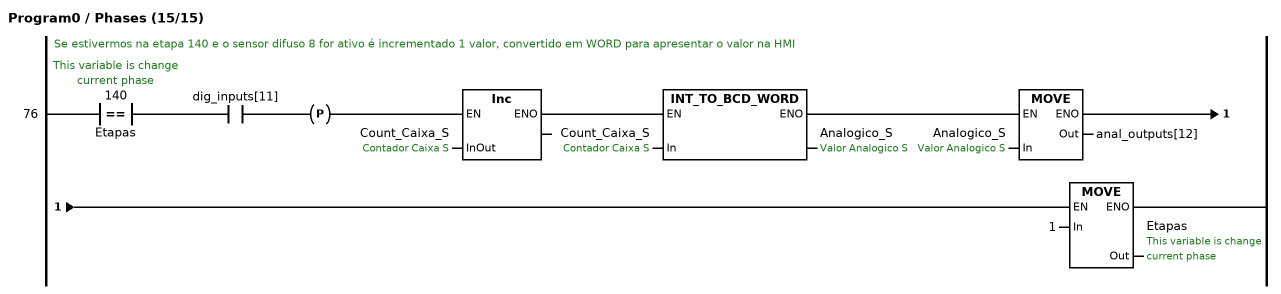
(* Rung 76: Se estivermos na etapa 140 e o sensor difuso 8 for ativo é incrementado 1 valor, convertido em WORD para apresentar o valor na HMI *)
_e8(CLK := (140 = Etapas) AND dig_inputs[11]);
IF _e8.Q THEN
    Inc(InOut := Count_Caixa_S);
    Analogico_S := INT_TO_BCD_WORD(In := Count_Caixa_S);
    anal_outputs[12] := Analogico_S;
    Etapas := 1;
END_IF;

(* Section Outputs: ladder, written here as Structured Text *)

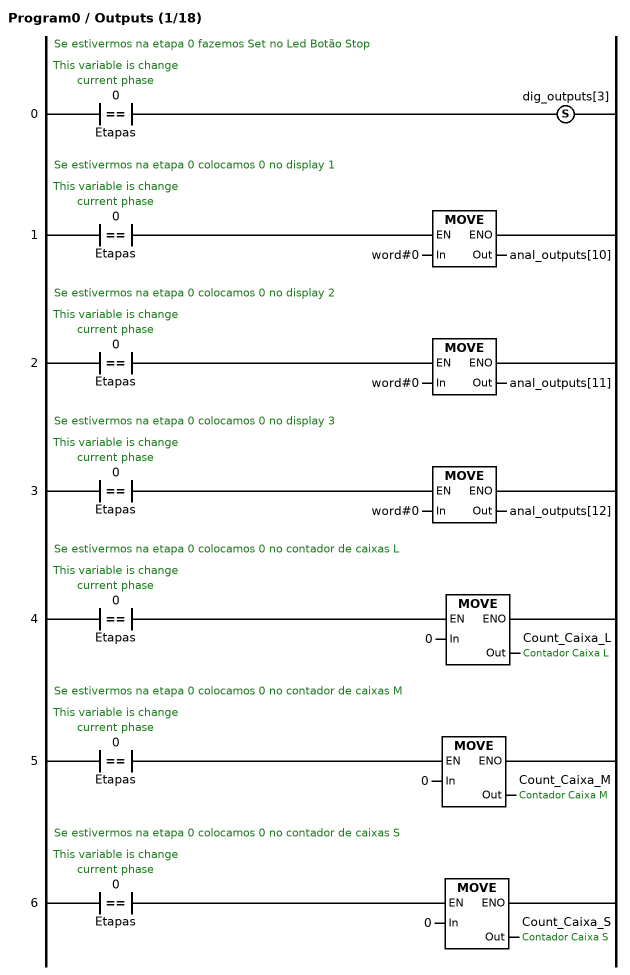
(* Rung 0: Se estivermos na etapa 0 fazemos Set no Led Botão Stop *)
IF 0 = Etapas THEN dig_outputs[3] := TRUE; END_IF;
(* Rung 1: Se estivermos na etapa 0 colocamos 0 no display 1 *)
IF 0 = Etapas THEN anal_outputs[10] := word#0; END_IF;
(* Rung 2: Se estivermos na etapa 0 colocamos 0 no display 2 *)
IF 0 = Etapas THEN anal_outputs[11] := word#0; END_IF;
(* Rung 3: Se estivermos na etapa 0 colocamos 0 no display 3 *)
IF 0 = Etapas THEN anal_outputs[12] := word#0; END_IF;
(* Rung 4: Se estivermos na etapa 0 colocamos 0 no contador de caixas L *)
IF 0 = Etapas THEN Count_Caixa_L := 0; END_IF;
(* Rung 5: Se estivermos na etapa 0 colocamos 0 no contador de caixas M *)
IF 0 = Etapas THEN Count_Caixa_M := 0; END_IF;
(* Rung 6: Se estivermos na etapa 0 colocamos 0 no contador de caixas S *)
IF 0 = Etapas THEN Count_Caixa_S := 0; END_IF;

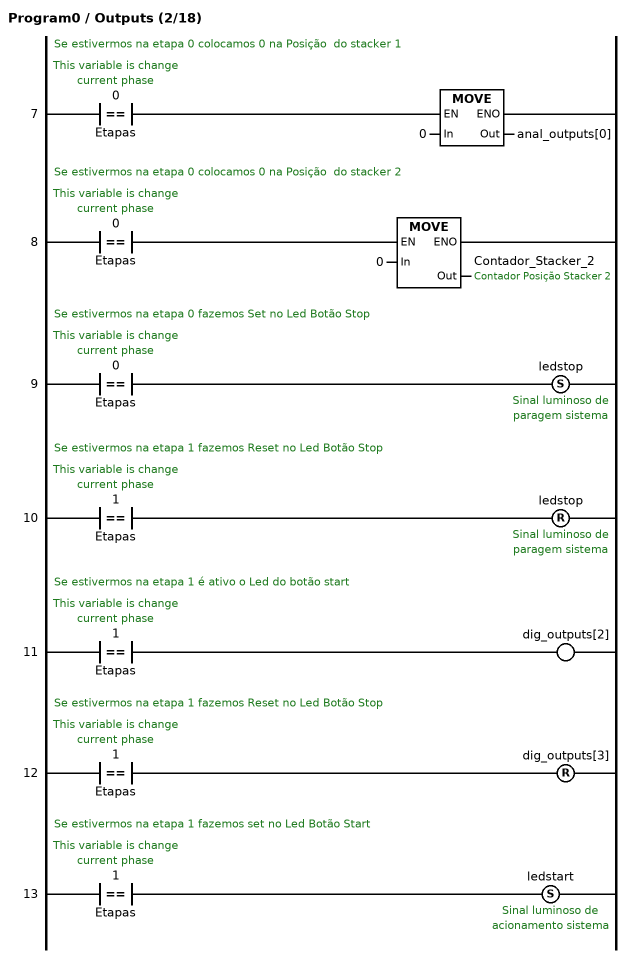
(* Rung 7: Se estivermos na etapa 0 colocamos 0 na Posição  do stacker 1 *)
IF 0 = Etapas THEN anal_outputs[0] := 0; END_IF;
(* Rung 8: Se estivermos na etapa 0 colocamos 0 na Posição  do stacker 2 *)
IF 0 = Etapas THEN Contador_Stacker_2 := 0; END_IF;
(* Rung 9: Se estivermos na etapa 0 fazemos Set no Led Botão Stop *)
IF 0 = Etapas THEN ledstop := TRUE; END_IF;
(* Rung 10: Se estivermos na etapa 1 fazemos Reset no Led Botão Stop *)
IF 1 = Etapas THEN ledstop := FALSE; END_IF;
(* Rung 11: Se estivermos na etapa 1 é ativo o Led do botão start *)
dig_outputs[2] := 1 = Etapas;
(* Rung 12: Se estivermos na etapa 1 fazemos Reset no Led Botão Stop *)
IF 1 = Etapas THEN dig_outputs[3] := FALSE; END_IF;
(* Rung 13: Se estivermos na etapa 1 fazemos set no Led Botão Start *)
IF 1 = Etapas THEN ledstart := TRUE; END_IF;

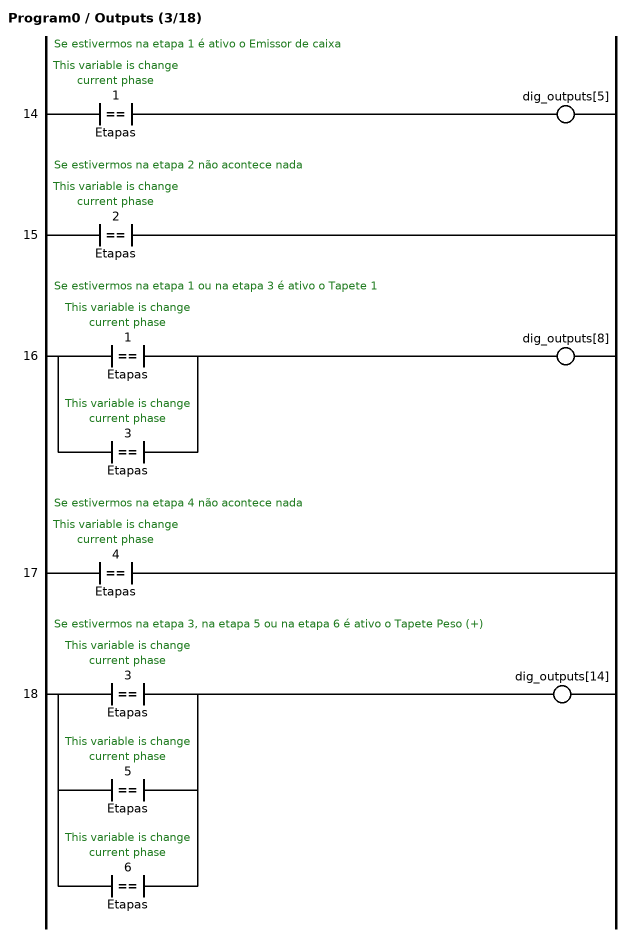
(* Rung 14: Se estivermos na etapa 1 é ativo o Emissor de caixa *)
dig_outputs[5] := 1 = Etapas;
(* Rung 15: Se estivermos na etapa 2 não acontece nada *)
(* drawn but driving nothing: Etapas *)
(* Rung 16: Se estivermos na etapa 1 ou na etapa 3 é ativo o Tapete 1 *)
dig_outputs[8] := (1 = Etapas) OR (3 = Etapas);
(* Rung 17: Se estivermos na etapa 4 não acontece nada *)
(* drawn but driving nothing: Etapas *)
(* Rung 18: Se estivermos na etapa 3, na etapa 5 ou na etapa 6 é ativo o Tapete Peso (+) *)
dig_outputs[14] := (3 = Etapas) OR (5 = Etapas) OR (6 = Etapas);

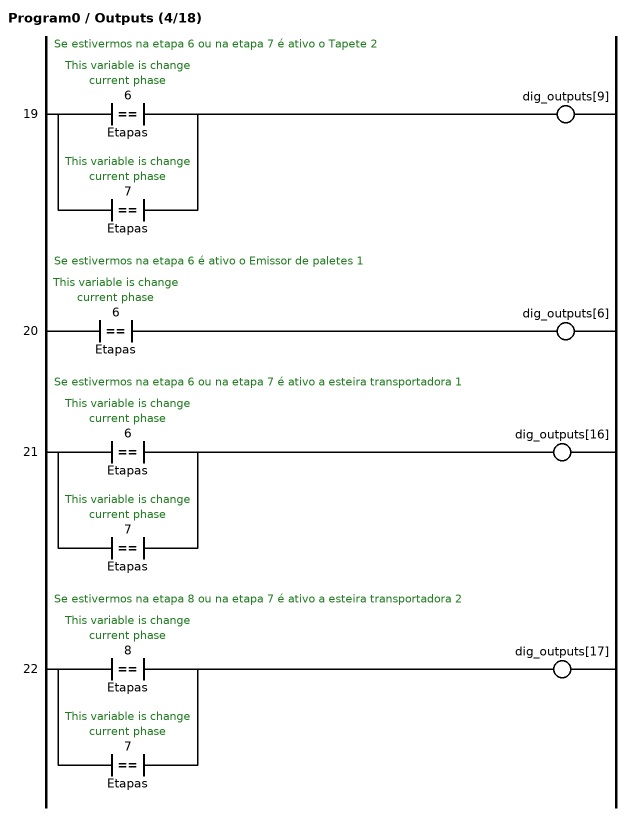
(* Rung 19: Se estivermos na etapa 6 ou na etapa 7 é ativo o Tapete 2 *)
dig_outputs[9] := (6 = Etapas) OR (7 = Etapas);
(* Rung 20: Se estivermos na etapa 6 é ativo o Emissor de paletes 1 *)
dig_outputs[6] := 6 = Etapas;
(* Rung 21: Se estivermos na etapa 6 ou na etapa 7 é ativo a esteira transportadora 1 *)
dig_outputs[16] := (6 = Etapas) OR (7 = Etapas);
(* Rung 22: Se estivermos na etapa 8 ou na etapa 7 é ativo a esteira transportadora 2 *)
dig_outputs[17] := (8 = Etapas) OR (7 = Etapas);

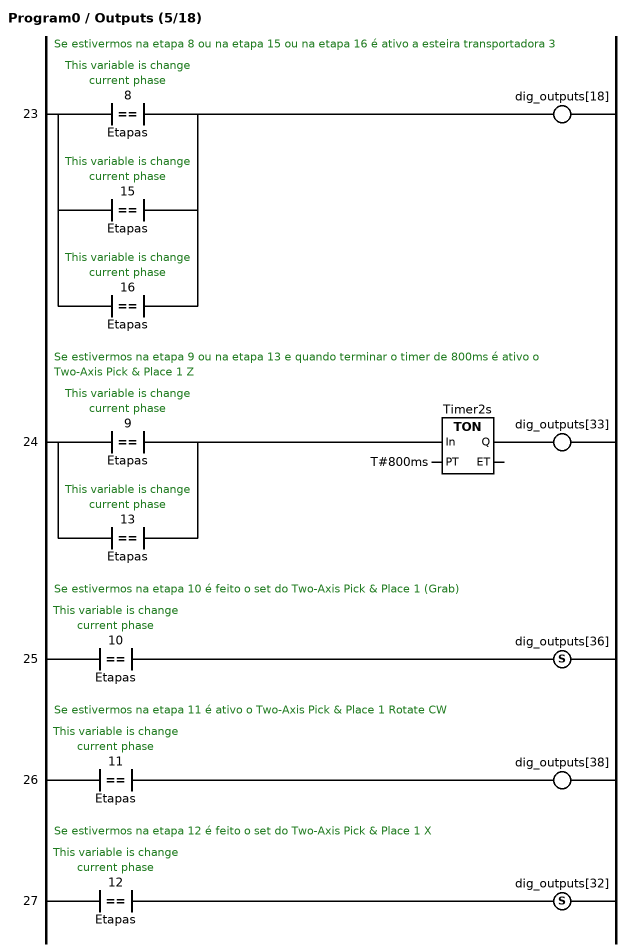
(* Rung 23: Se estivermos na etapa 8 ou na etapa 15 ou na etapa 16 é ativo a esteira transportadora 3 *)
dig_outputs[18] := (8 = Etapas) OR (15 = Etapas) OR (16 = Etapas);
(* Rung 24: Se estivermos na etapa 9 ou na etapa 13 e quando terminar o timer de 800ms é ativo o Two-Axis Pick & Place 1 Z *)
Timer2s(In := (9 = Etapas) OR (13 = Etapas), PT := T#800ms);
dig_outputs[33] := Timer2s.Q;
(* Rung 25: Se estivermos na etapa 10 é feito o set do Two-Axis Pick & Place 1 (Grab) *)
IF 10 = Etapas THEN dig_outputs[36] := TRUE; END_IF;
(* Rung 26: Se estivermos na etapa 11 é ativo o Two-Axis Pick & Place 1 Rotate CW *)
dig_outputs[38] := 11 = Etapas;
(* Rung 27: Se estivermos na etapa 12 é feito o set do Two-Axis Pick & Place 1 X *)
IF 12 = Etapas THEN dig_outputs[32] := TRUE; END_IF;

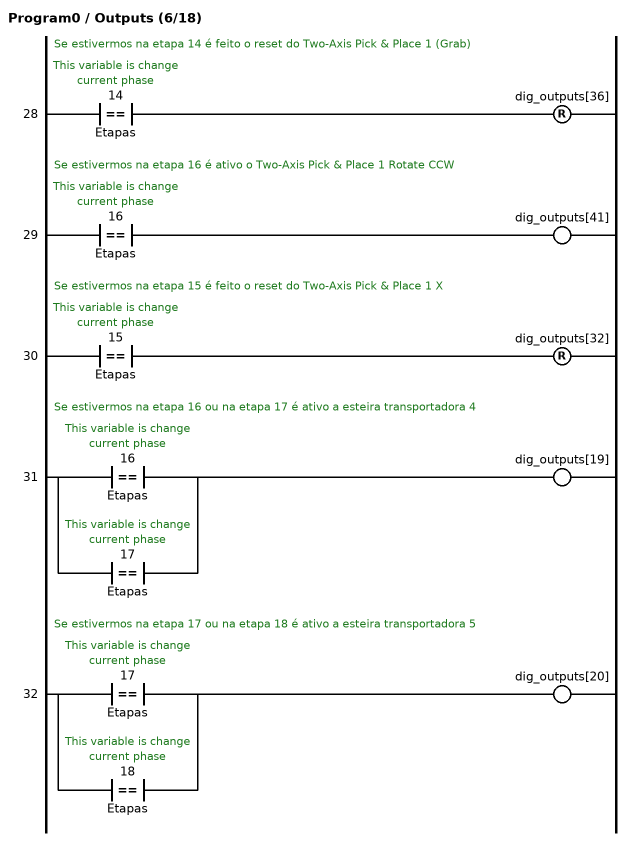
(* Rung 28: Se estivermos na etapa 14 é feito o reset do Two-Axis Pick & Place 1 (Grab) *)
IF 14 = Etapas THEN dig_outputs[36] := FALSE; END_IF;
(* Rung 29: Se estivermos na etapa 16 é ativo o Two-Axis Pick & Place 1 Rotate CCW *)
dig_outputs[41] := 16 = Etapas;
(* Rung 30: Se estivermos na etapa 15 é feito o reset do Two-Axis Pick & Place 1 X *)
IF 15 = Etapas THEN dig_outputs[32] := FALSE; END_IF;
(* Rung 31: Se estivermos na etapa 16 ou na etapa 17 é ativo a esteira transportadora 4 *)
dig_outputs[19] := (16 = Etapas) OR (17 = Etapas);
(* Rung 32: Se estivermos na etapa 17 ou na etapa 18 é ativo a esteira transportadora 5 *)
dig_outputs[20] := (17 = Etapas) OR (18 = Etapas);

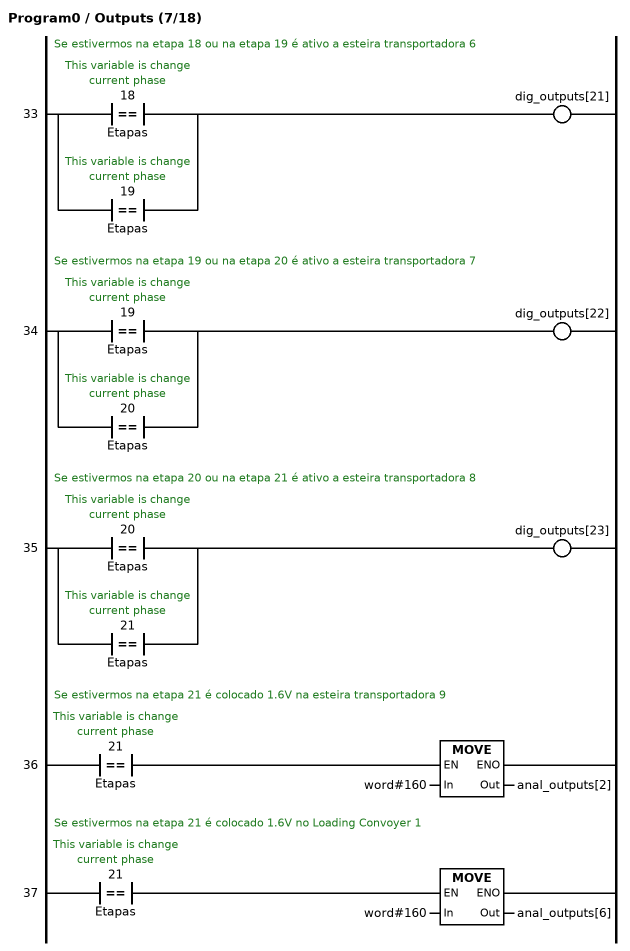
(* Rung 33: Se estivermos na etapa 18 ou na etapa 19 é ativo a esteira transportadora 6 *)
dig_outputs[21] := (18 = Etapas) OR (19 = Etapas);
(* Rung 34: Se estivermos na etapa 19 ou na etapa 20 é ativo a esteira transportadora 7 *)
dig_outputs[22] := (19 = Etapas) OR (20 = Etapas);
(* Rung 35: Se estivermos na etapa 20 ou na etapa 21 é ativo a esteira transportadora 8 *)
dig_outputs[23] := (20 = Etapas) OR (21 = Etapas);
(* Rung 36: Se estivermos na etapa 21 é colocado 1.6V na esteira transportadora 9 *)
IF 21 = Etapas THEN anal_outputs[2] := word#160; END_IF;
(* Rung 37: Se estivermos na etapa 21 é colocado 1.6V no Loading Convoyer 1 *)
IF 21 = Etapas THEN anal_outputs[6] := word#160; END_IF;

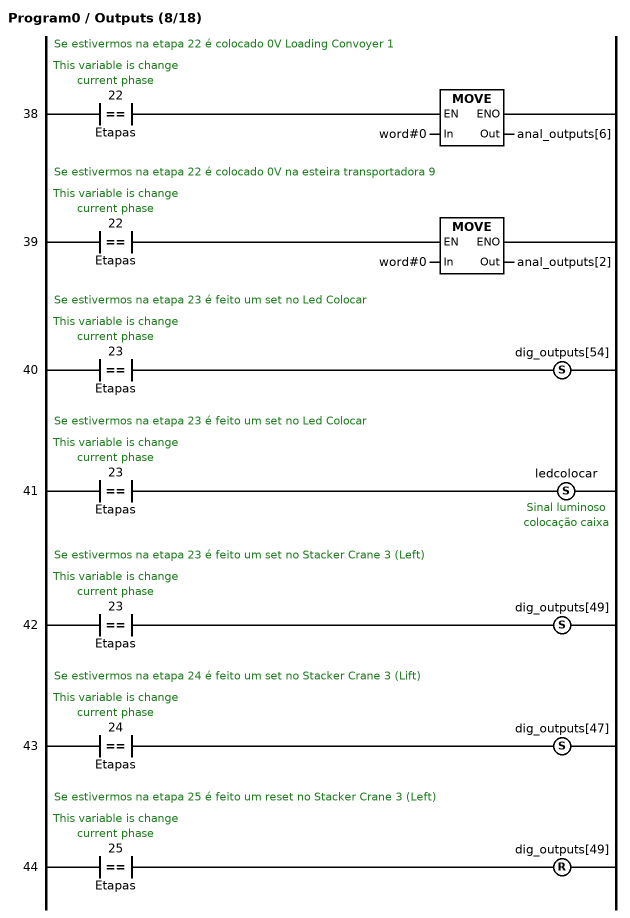
(* Rung 38: Se estivermos na etapa 22 é colocado 0V Loading Convoyer 1 *)
IF 22 = Etapas THEN anal_outputs[6] := word#0; END_IF;
(* Rung 39: Se estivermos na etapa 22 é colocado 0V na esteira transportadora 9 *)
IF 22 = Etapas THEN anal_outputs[2] := word#0; END_IF;
(* Rung 40: Se estivermos na etapa 23 é feito um set no Led Colocar *)
IF 23 = Etapas THEN dig_outputs[54] := TRUE; END_IF;
(* Rung 41: Se estivermos na etapa 23 é feito um set no Led Colocar *)
IF 23 = Etapas THEN ledcolocar := TRUE; END_IF;
(* Rung 42: Se estivermos na etapa 23 é feito um set no Stacker Crane 3 (Left) *)
IF 23 = Etapas THEN dig_outputs[49] := TRUE; END_IF;
(* Rung 43: Se estivermos na etapa 24 é feito um set no Stacker Crane 3 (Lift) *)
IF 24 = Etapas THEN dig_outputs[47] := TRUE; END_IF;
(* Rung 44: Se estivermos na etapa 25 é feito um reset no Stacker Crane 3 (Left) *)
IF 25 = Etapas THEN dig_outputs[49] := FALSE; END_IF;

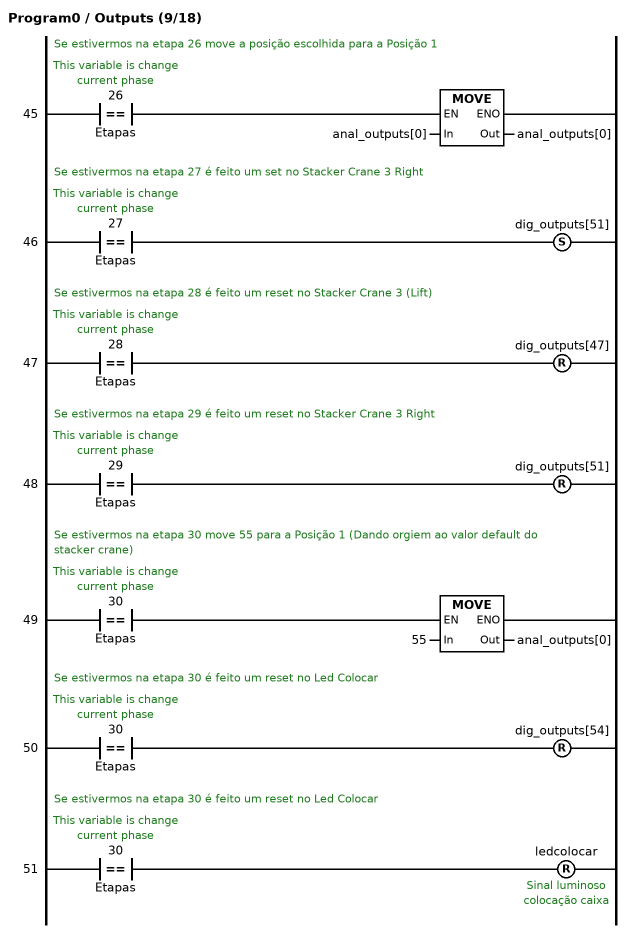
(* Rung 45: Se estivermos na etapa 26 move a posição escolhida para a Posição 1 *)
IF 26 = Etapas THEN anal_outputs[0] := anal_outputs[0]; END_IF;
(* Rung 46: Se estivermos na etapa 27 é feito um set no Stacker Crane 3 Right *)
IF 27 = Etapas THEN dig_outputs[51] := TRUE; END_IF;
(* Rung 47: Se estivermos na etapa 28 é feito um reset no Stacker Crane 3 (Lift) *)
IF 28 = Etapas THEN dig_outputs[47] := FALSE; END_IF;
(* Rung 48: Se estivermos na etapa 29 é feito um reset no Stacker Crane 3 Right *)
IF 29 = Etapas THEN dig_outputs[51] := FALSE; END_IF;
(* Rung 49: Se estivermos na etapa 30 move 55 para a Posição 1 (Dando orgiem ao valor default do stacker crane) *)
IF 30 = Etapas THEN anal_outputs[0] := 55; END_IF;
(* Rung 50: Se estivermos na etapa 30 é feito um reset no Led Colocar *)
IF 30 = Etapas THEN dig_outputs[54] := FALSE; END_IF;
(* Rung 51: Se estivermos na etapa 30 é feito um reset no Led Colocar *)
IF 30 = Etapas THEN ledcolocar := FALSE; END_IF;

